{attribute 'qualified_only'}
VAR_GLOBAL
	RestartSAFETY AT%Q* : BOOL;
END_VAR

(* stored: Version 1.1.0.1, ProductVersion 3.1.4024.3
   GVL GVL_SAFETY: Id {cb20a1ae-5c2d-4093-bc98-22c75603def5} *)
